{attribute 'GeneratedUsingTerminal: EK1100-0000-0018'}
{attribute addProperty BoxType "EK1100-0000-0018"}
{attribute addProperty Id "Beckhoff_ER4xxxEK1122Beckhoff_ER4xxxEK1122_5C895096112"}
{attribute addProperty CRC "2038098869"}
{attribute addProperty Size "112"}
TYPE Beckhoff_ER4xxx_797AEBB5 EXTENDS EK1100_1FC0878B :
STRUCT
	{attribute addProperty Name "Beckhoff ER4xxxEK1122"}
	{attribute addProperty PreviousPort "Beckhoff ER4xxx : B"}
	Beckhoff_ER4xxxEK1122 : Beckhoff_ER4xxxEK1122_5C895096;
END_STRUCT
END_TYPE

(* stored: Version 1.2.0.0, ProductVersion 3.1.4024.9
   DUT Beckhoff_ER4xxx_797AEBB5: Id {2286e961-5058-433b-8909-64736ba97679} *)
